// TIA Portal V19 export
TYPE "LEXCHANGETRAY_typeRollerVfdContronNodeCommandConfiguration"
// highVel: Real
// lowVel: Real
// direction: DInt
// sinaCommandConfiguration: LBC_typeSinaSpeedCommandConfiguration
// stored: Access Published
   STRUCT
      highVel : Real;
      lowVel { S7_SetPoint := 'True'} : Real;
      direction : DInt := 1;
      sinaCommandConfiguration : "LBC_typeSinaSpeedCommandConfiguration";
   END_STRUCT;
END_TYPE
